{attribute 'qualified_only'}
VAR_GLOBAL
	Start : BOOL;
	Stopp : BOOL := FALSE;
	NotStopp : BOOL := TRUE;
	Fehler			: BOOL;
	Weiter			: BOOL;
	DiagnoseRequested: BOOL;
END_VAR

(* stored: Version 1.1.0.1
   GVL GVL: Id {7ea246ce-2a6d-4b87-aac6-827fdf3c548d} *)
